TYPE ST_RS485ComDeviceStatus :
STRUCT
	diID			:DINT;			
	sState			:STRING;
	bCOM			:BOOL;					(*Zeigt die Kommunikation an *)
	bStartupDone	:BOOL;
	bError			:BOOL;
	
	(* Vorbehalt für Taster *)
	lrTemp			:LREAL;						(* Temperatur Sensor	*)
	lrRhd			:LREAL;						(* Luftfeuchtigkeit Sensor	*)
	lrBrs			:LREAL;						(* Helligkeit Sensor *)
		
	dwChanges		:DWORD;				
END_STRUCT
END_TYPE

(* stored: Version 1.1.0.1, ProductVersion 3.1.4024.12
   DUT ST_RS485ComDeviceStatus: Id {d6fdbac6-ff1d-47fa-9166-63340e1d4984} *)
